// TIA Portal V18 export
TYPE "MEStoPLC_Common"
// stored: IsFailsafeCompliant false
   STRUCT
      "M-MesOnline" : Bool;   // MES在线信号=1，常为1，0=Offline
      "M-HeartBeat" : Bool;   // MES心跳信号，频率5S，PLC10S延迟判定报警
      Reserve : Array[1..197] of Byte;   // Common交互预留
   END_STRUCT;
END_TYPE
